LIN {X 0,Y 64.224,Z 923.35,A -85,B 0,C 180,E1 -22998.896,E2 -22998.896} C_VEL
LIN {X 0,Y 56.678,Z 935.443,A -85,B 0,C 180,E1 -23073.735,E2 -23073.735} C_VEL
LIN {X 0,Y 46.519,Z 939.9,A -85,B 0,C 180,E1 -23092.995,E2 -23092.995} C_VEL
LIN {X 0,Y 43.445,Z 942.454,A -85,B 0,C 180,E1 -23118.042,E2 -23118.042} C_VEL
LIN {X 0,Y 44.609,Z 942.986,A -85,B 0,C 180,E1 -23129.996,E2 -23129.996} C_VEL
LIN {X 0,Y 43.43,Z 941.643,A -85,B 0,C 180,E1 -23151.61,E2 -23151.61} C_VEL
LIN {X 0,Y 48.607,Z 938.528,A -85,B 0,C 180,E1 -23174.374,E2 -23174.374} C_VEL
LIN {X 0,Y 60.109,Z 933.405,A -85,B 0,C 180,E1 -23191.831,E2 -23191.831} C_VEL
LIN {X 0,Y 75.231,Z 926.324,A -85,B 0,C 180,E1 -23203.114,E2 -23203.114} C_VEL
LIN {X 0,Y 91.338,Z 917.638,A -85,B 0,C 180,E1 -23210.125,E2 -23210.125} C_VEL
LIN {X 0,Y 107.429,Z 907.425,A -85,B 0,C 180,E1 -23214.772,E2 -23214.772} C_VEL
LIN {X 0,Y 123.058,Z 895.783,A -85,B 0,C 180,E1 -23217.955,E2 -23217.955} C_VEL
LIN {X 0,Y 137.979,Z 882.698,A -85,B 0,C 180,E1 -23220.243,E2 -23220.243} C_VEL
LIN {X 0,Y 143.407,Z 877.402,A -85,B 0,C 180,E1 -23220.953,E2 -23220.953} C_VEL
LIN {X 0,Y 146.706,Z 873.855,A -85,B 0,C 180,E1 -23221.746,E2 -23221.746} C_VEL
LIN {X 0,Y 154.441,Z 864.839,A -85,B 0,C 180,E1 -23224.886,E2 -23224.886} C_VEL
LIN {X 0,Y 157.162,Z 861.551,A -85,B 0,C 180,E1 -23225.398,E2 -23225.398} C_VEL
LIN {X 0,Y 159.112,Z 859.162,A -85,B 0,C 180,E1 -23225.559,E2 -23225.559} C_VEL
LIN {X 0,Y 147.111,Z 872.273,A -85,B 0,C 180,E1 -23227.119,E2 -23227.119} C_VEL
LIN {X 0,Y 133.663,Z 884.599,A -85,B 0,C 180,E1 -23229.106,E2 -23229.106} C_VEL
LIN {X 0,Y 119.428,Z 895.511,A -85,B 0,C 180,E1 -23231.619,E2 -23231.619} C_VEL
LIN {X 0,Y 103.925,Z 905.376,A -85,B 0,C 180,E1 -23235.058,E2 -23235.058} C_VEL
LIN {X 0,Y 88.18,Z 913.572,A -85,B 0,C 180,E1 -23239.765,E2 -23239.765} C_VEL
LIN {X 0,Y 72.637,Z 920.099,A -85,B 0,C 180,E1 -23246.53,E2 -23246.53} C_VEL
LIN {X 0,Y 57.671,Z 925.065,A -85,B 0,C 180,E1 -23257.111,E2 -23257.111} C_VEL
LIN {X 0,Y 45.511,Z 928.191,A -85,B 0,C 180,E1 -23273.621,E2 -23273.621} C_VEL
LIN {X 0,Y 38.534,Z 929.646,A -85,B 0,C 180,E1 -23298.024,E2 -23298.024} C_VEL
LIN {X 0,Y 38.932,Z 929.594,A -85,B 0,C 180,E1 -23324.886,E2 -23324.886} C_VEL
LIN {X 0,Y 46.571,Z 927.983,A -85,B 0,C 180,E1 -23348.512,E2 -23348.512} C_VEL
LIN {X 0,Y 53.609,Z 926.212,A -85,B 0,C 180,E1 -23358.855,E2 -23358.855} C_VEL
LIN {X 0,Y 46.893,Z 936.123,A -85,B 0,C 180,E1 -23432.895,E2 -23432.895} C_VEL
LIN {X 0,Y 37.076,Z 939.865,A -85,B 0,C 180,E1 -23457.355,E2 -23457.355} C_VEL
LIN {X 0,Y 36.08,Z 941.56,A -85,B 0,C 180,E1 -23486.01,E2 -23486.01} C_VEL
LIN {X 0,Y 36.51,Z 941.691,A -85,B 0,C 180,E1 -23489.996,E2 -23489.996} C_VEL
LIN {X 0,Y 36.049,Z 940.202,A -85,B 0,C 180,E1 -23518.127,E2 -23518.127} C_VEL
LIN {X 0,Y 44.22,Z 936.762,A -85,B 0,C 180,E1 -23544.483,E2 -23544.483} C_VEL
LIN {X 0,Y 58.26,Z 931.432,A -85,B 0,C 180,E1 -23560.711,E2 -23560.711} C_VEL
LIN {X 0,Y 75.069,Z 924.088,A -85,B 0,C 180,E1 -23570.26,E2 -23570.26} C_VEL
LIN {X 0,Y 92.215,Z 915.153,A -85,B 0,C 180,E1 -23575.95,E2 -23575.95} C_VEL
LIN {X 0,Y 108.984,Z 904.705,A -85,B 0,C 180,E1 -23579.651,E2 -23579.651} C_VEL
LIN {X 0,Y 125.067,Z 892.807,A -85,B 0,C 180,E1 -23582.135,E2 -23582.135} C_VEL
LIN {X 0,Y 140.31,Z 879.415,A -85,B 0,C 180,E1 -23583.942,E2 -23583.942} C_VEL
LIN {X 0,Y 154.151,Z 864.999,A -85,B 0,C 180,E1 -23585.164,E2 -23585.164} C_VEL
LIN {X 0,Y 157.162,Z 861.551,A -85,B 0,C 180,E1 -23585.398,E2 -23585.398} C_VEL
LIN {X 0,Y 160.605,Z 862.838,A -85,B 0,C 180,E1 -23585.68,E2 -23585.68} C_VEL
LIN {X 0,Y 160.605,Z 899.419,A -85,B 0,C 180,E1 -23585.68,E2 -23585.68} C_VEL
LIN {X 0,Y 133.78,Z 899.419,A -85,B 0,C 180,E1 -23585.842,E2 -23585.842} C_VEL
LIN {X 0,Y 131.781,Z 897.419,A -85,B 0,C 180,E1 -23585.857,E2 -23585.857} C_VEL
LIN {X 0,Y 131.781,Z 890.637,A -85,B 0,C 180,E1 -23585.857,E2 -23585.857} C_VEL
LIN {X 0,Y 128.747,Z 889.015,A -85,B 0,C 180,E1 -23586.262,E2 -23586.262} C_VEL
LIN {X 0,Y 113.272,Z 899.981,A -85,B 0,C 180,E1 -23588.658,E2 -23588.658} C_VEL
LIN {X 0,Y 98.007,Z 908.899,A -85,B 0,C 180,E1 -23591.663,E2 -23591.663} C_VEL
LIN {X 0,Y 82.129,Z 916.445,A -85,B 0,C 180,E1 -23595.902,E2 -23595.902} C_VEL
LIN {X 0,Y 65.931,Z 922.544,A -85,B 0,C 180,E1 -23602.327,E2 -23602.327} C_VEL
LIN {X 0,Y 50.087,Z 927.092,A -85,B 0,C 180,E1 -23613.033,E2 -23613.033} C_VEL
LIN {X 0,Y 37.029,Z 929.861,A -85,B 0,C 180,E1 -23631.613,E2 -23631.613} C_VEL
LIN {X 0,Y 30.14,Z 930.987,A -85,B 0,C 180,E1 -23662.38,E2 -23662.38} C_VEL
LIN {X 0,Y 32.699,Z 930.614,A -85,B 0,C 180,E1 -23695.352,E2 -23695.352} C_VEL
LIN {X 0,Y 42.954,Z 928.761,A -85,B 0,C 180,E1 -23719.1,E2 -23719.1} C_VEL
LIN {X 0,Y 37.126,Z 936.508,A -85,B 0,C 180,E1 -23791.659,E2 -23791.659} C_VEL
LIN {X 0,Y 28.168,Z 939.404,A -85,B 0,C 180,E1 -23822.538,E2 -23822.538} C_VEL
LIN {X 0,Y 28.38,Z 940.39,A -85,B 0,C 180,E1 -23849.994,E2 -23849.994} C_VEL
LIN {X 0,Y 29.342,Z 938.756,A -85,B 0,C 180,E1 -23887.826,E2 -23887.826} C_VEL
LIN {X 0,Y 40.69,Z 935.195,A -85,B 0,C 180,E1 -23915.383,E2 -23915.383} C_VEL
LIN {X 0,Y 56.956,Z 929.73,A -85,B 0,C 180,E1 -23929.427,E2 -23929.427} C_VEL
LIN {X 0,Y 74.787,Z 922.416,A -85,B 0,C 180,E1 -23936.937,E2 -23936.937} C_VEL
LIN {X 0,Y 92.169,Z 913.708,A -85,B 0,C 180,E1 -23941.245,E2 -23941.245} C_VEL
LIN {X 0,Y 109.259,Z 903.355,A -85,B 0,C 180,E1 -23944.084,E2 -23944.084} C_VEL
LIN {X 0,Y 125.66,Z 891.466,A -85,B 0,C 180,E1 -23945.966,E2 -23945.966} C_VEL
LIN {X 0,Y 128.747,Z 889.015,A -85,B 0,C 180,E1 -23946.262,E2 -23946.262} C_VEL
LIN {X 0,Y 129.02,Z 890.99,A -85,B 0,C 180,E1 -23947.284,E2 -23947.284} C_VEL
LIN {X 0,Y 129.02,Z 920.241,A -85,B 0,C 180,E1 -23947.284,E2 -23947.284} C_VEL
LIN {X 0,Y 101.361,Z 920.241,A -85,B 0,C 180,E1 -23946.407,E2 -23946.407} C_VEL
LIN {X 0,Y 99.366,Z 918.241,A -85,B 0,C 180,E1 -23946.325,E2 -23946.325} C_VEL
LIN {X 0,Y 99.366,Z 911.941,A -85,B 0,C 180,E1 -23946.325,E2 -23946.325} C_VEL
LIN {X 0,Y 96.842,Z 910.105,A -85,B 0,C 180,E1 -23947.026,E2 -23947.026} C_VEL
LIN {X 0,Y 80.32,Z 917.712,A -85,B 0,C 180,E1 -23950.457,E2 -23950.457} C_VEL
LIN {X 0,Y 63.347,Z 923.812,A -85,B 0,C 180,E1 -23955.682,E2 -23955.682} C_VEL
LIN {X 0,Y 46.249,Z 928.359,A -85,B 0,C 180,E1 -23964.778,E2 -23964.778} C_VEL
LIN {X 0,Y 31.218,Z 931.127,A -85,B 0,C 180,E1 -23982.561,E2 -23982.561} C_VEL
LIN {X 0,Y 22.335,Z 932.251,A -85,B 0,C 180,E1 -24019.692,E2 -24019.692} C_VEL
LIN {X 0,Y 25.778,Z 931.878,A -85,B 0,C 180,E1 -24062.897,E2 -24062.897} C_VEL
LIN {X 0,Y 32.06,Z 931.05,A -85,B 0,C 180,E1 -24079.493,E2 -24079.493} C_VEL
LIN {X 0,Y 27.354,Z 936.612,A -85,B 0,C 180,E1 -24149.665,E2 -24149.665} C_VEL
LIN {X 0,Y 19.648,Z 938.787,A -85,B 0,C 180,E1 -24195.251,E2 -24195.251} C_VEL
LIN {X 0,Y 20.211,Z 939.084,A -85,B 0,C 180,E1 -24209.992,E2 -24209.992} C_VEL
LIN {X 0,Y 23.332,Z 937.425,A -85,B 0,C 180,E1 -24260.466,E2 -24260.466} C_VEL
LIN {X 0,Y 37.965,Z 933.849,A -85,B 0,C 180,E1 -24287,E2 -24287} C_VEL
LIN {X 0,Y 56.05,Z 928.37,A -85,B 0,C 180,E1 -24297.958,E2 -24297.958} C_VEL
LIN {X 0,Y 74.107,Z 921.381,A -85,B 0,C 180,E1 -24303.269,E2 -24303.269} C_VEL
LIN {X 0,Y 92.572,Z 912.447,A -85,B 0,C 180,E1 -24306.458,E2 -24306.458} C_VEL
LIN {X 0,Y 96.842,Z 910.105,A -85,B 0,C 180,E1 -24307.026,E2 -24307.026} C_VEL
LIN {X 0,Y 89.772,Z 913.57,A -85,B 0,C 180,E1 -24308.543,E2 -24308.543} C_VEL
LIN {X 0,Y 80.959,Z 917.583,A -85,B 0,C 180,E1 -24309.313,E2 -24309.313} C_VEL
LIN {X 0,Y 69.735,Z 922.242,A -85,B 0,C 180,E1 -24308.858,E2 -24308.858} C_VEL
LIN {X 0,Y 52.558,Z 928.213,A -85,B 0,C 180,E1 -24305.644,E2 -24305.644} C_VEL
LIN {X 0,Y 33.026,Z 933.368,A -85,B 0,C 180,E1 -24297.414,E2 -24297.414} C_VEL
LIN {X 0,Y 15.594,Z 936.641,A -85,B 0,C 180,E1 -24269.153,E2 -24269.153} C_VEL
LIN {X 0,Y 12.008,Z 937.767,A -85,B 0,C 180,E1 -24207.337,E2 -24207.337} C_VEL
LIN {X 0,Y 17.736,Z 936.397,A -85,B 0,C 180,E1 -24145.003,E2 -24145.003} C_VEL
LIN {X 0,Y 21.136,Z 933.014,A -85,B 0,C 180,E1 -24079.855,E2 -24079.855} C_VEL
LIN {X 0,Y 14.243,Z 933.555,A -85,B 0,C 180,E1 -24021.94,E2 -24021.94} C_VEL
LIN {X 0,Y 24.078,Z 932.697,A -85,B 0,C 180,E1 -23973.859,E2 -23973.859} C_VEL
LIN {X 0,Y 40.732,Z 930.192,A -85,B 0,C 180,E1 -23956.808,E2 -23956.808} C_VEL
LIN {X 0,Y 58.776,Z 925.922,A -85,B 0,C 180,E1 -23949.384,E2 -23949.384} C_VEL
LIN {X 0,Y 63.61,Z 924.528,A -85,B 0,C 180,E1 -23948.018,E2 -23948.018} C_VEL
LIN {X 0,Y 52.558,Z 928.213,A -85,B 0,C 180,E1 -23945.644,E2 -23945.644} C_VEL
LIN {X 0,Y 45.291,Z 930.231,A -85,B 0,C 180,E1 -23944.636,E2 -23944.636} C_VEL
LIN {X 0,Y 35.562,Z 932.166,A -85,B 0,C 180,E1 -23945.91,E2 -23945.91} C_VEL
LIN {X 0,Y 17.444,Z 934.242,A -85,B 0,C 180,E1 -23959.124,E2 -23959.124} C_VEL
LIN {X 0,Y 16.348,Z 934.308,A -85,B 0,C 180,E1 -23960.73,E2 -23960.73} C_VEL
LIN {X 0,Y 6.875,Z 934.805,A -85,B 0,C 180,E1 -24055.895,E2 -24055.895} C_VEL
LIN {X 0,Y 10.26,Z 934.714,A -85,B 0,C 180,E1 -24084.198,E2 -24084.198} C_VEL
LIN {X 0,Y 8.178,Z 935.951,A -85,B 0,C 180,E1 -24131.931,E2 -24131.931} C_VEL
LIN {X 0,Y 3.799,Z 936.459,A -85,B 0,C 180,E1 -24209.957,E2 -24209.957} C_VEL
LIN {X 0,Y 18.57,Z 934.691,A -85,B 0,C 180,E1 -24306.191,E2 -24306.191} C_VEL
LIN {X 0,Y 27.45,Z 933.255,A -85,B 0,C 180,E1 -24310.46,E2 -24310.46} C_VEL
LIN {X 0,Y 16.348,Z 934.308,A -85,B 0,C 180,E1 -24320.73,E2 -24320.73} C_VEL
LIN {X 0,Y 14.645,Z 936.304,A -85,B 0,C 180,E1 -24323.694,E2 -24323.694} C_VEL
LIN {X 0,Y 14.645,Z 1015.5,A -85,B 0,C 180,E1 -24323.694,E2 -24323.694} C_VEL
LIN {X 0,Y 14.645,Z 1015.5,A -85,B 0,C 180,E1 -24323.694,E2 -24323.694}

QRS_NEXT_CUT()

QRS_NEXT()
QRS_HOME()

END
